{attribute 'OPC.UA.DA.StructuredType' := '1'}
TYPE SNamedValue EXTENDS SValue :
STRUCT
	Name: STRING;
END_STRUCT
END_TYPE

(* stored: Version 1.1.0.1
   DUT SNamedValue: Id {37b3add2-6455-4754-a945-003725ab7ef3} *)
